// TwinCAT 3 PLC project PLC
// ProgramVersion: 3.1.4026.16
// libraries:
//   Tc2_Standard, * (Beckhoff Automation GmbH)
//   Tc2_System, * (Beckhoff Automation GmbH)
//   Tc3_Module, * (Beckhoff Automation GmbH)
// project tree:
//   / MAIN.TcPOU, PlcTask.TcTTO
//   POUs/ FB_ClkSignal.TcPOU
// real-time tasks:
//   TASK PlcTask: cycle T#10ms, priority 20, ADS port 350

CONFIGURATION PLC
    RESOURCE PLC ON TwinCAT3
        TASK PlcTask(INTERVAL := T#10ms, PRIORITY := 20);
        PROGRAM MAIN WITH PlcTask : MAIN;
    END_RESOURCE
END_CONFIGURATION

// ---- MAIN.TcPOU
PROGRAM MAIN
VAR

    bStart_Command : BOOL;
    fFreq_Setting  : REAL := 1.0; 

    bDigitalOutput AT %Q* : BOOL; 

    fbClockGen : FB_ClkSignal;
END_VAR

fbClockGen(
    IN_bStart := bStart_Command, 
    IN_fFrequency := fFreq_Setting, 
    OUT_Signal => bDigitalOutput
);

END_PROGRAM

// ---- POUs/FB_ClkSignal.TcPOU
FUNCTION_BLOCK FB_ClkSignal
VAR_INPUT
    IN_bStart : BOOL;       
    IN_fFrequency : REAL;   
END_VAR
VAR_OUTPUT
    OUT_Signal : BOOL;      
END_VAR
VAR
    timer : TON;            
    tHalfPeriod : TIME;     
END_VAR

IF IN_bStart AND IN_fFrequency > 0 THEN
    tHalfPeriod := REAL_TO_TIME((1.0 / IN_fFrequency) * 500.0);
    
    timer(IN := NOT timer.Q, PT := tHalfPeriod);
    
    IF timer.Q THEN
        OUT_Signal := NOT OUT_Signal;
    END_IF
ELSE
    OUT_Signal := FALSE;
    timer(IN := FALSE);
END_IF

END_FUNCTION_BLOCK
